Staubli VAL3: OMAC_Start.pgx

program OMAC_Start()
  local point l_pHere
begin

  //OMAC进程:Starting
  _nOmacStat=2
  logMsg("上位机手动操作：启动")
  // Task for cell manager
  if taskStatus("cellManager")>=0
    taskKill("cellManager")
  endIf
  wait(taskStatus("cellManager")<0)
  taskCreate "cellManager",100,cellManager()
  wait(taskStatus("cellManager")==1)

  delay(0)
end
